// TIA Portal V20 export
// export: Created 2025-12-01T14:56:22.0894666Z, ExportSetting None, DisplayName Totally Integrated Automation Portal, DisplayVersion V20 Update 3, DisplayName TIA Portal Openness, DisplayVersion V20 Update 3, DisplayName TIA Portal Version Control Interface, DisplayVersion V20 Update 3, DisplayName STEP 7 Professional, DisplayVersion V20 Update 3, DisplayName STEP 7 Safety, DisplayVersion V20 Update 2, DisplayName WinCC Basic/Comfort/Advanced, DisplayVersion V20 Update 3, DisplayName WinCC Professional, DisplayVersion V20 Update 3, DisplayName WinCC Unified, DisplayVersion V20 Update 3
TYPE "NDD_Interlock_Horquilla"
   STRUCT
      PosHorq_Bloqueo : Bool;   // La Horquilla esta en Bloqueo para ir a la Posicion IN (Hacia el Elevador)
      MovHorq_Bloqueada : Bool;
      OrdenDeSalida : Bool;   // Orden de la Salida de la Paleta de la Horquilla
      FinOrdenDeSalida : Bool;
      DejarCarga_EntradaHorq : Bool;
      DejadaCarga_EntradaHorq : Bool;   // Aviso de Dejar la Paleta en la Horquilla
      RecogerCarga_SalidaHorq : Bool;   // Aviso de Recoger la Paleta de la Horquilla
      RecogidaCarga_SalidaHorq : Bool;
      AVTF_EntradaHorq : Bool;   // Aviso de Entrada de la Paleta en la Horquilla
      PTF_EntradaHorq : Bool;   // Permiso de Entrada de la Paleta en la Horquilla
      FTF_EntradaHorq : Bool;   // Fin de la Entrada de la Paleta en la Horquilla
      AVTF_SalidaHorq : Bool;   // Aviso de Salida de la Paleta en la Horquilla
      PTF_SalidaHorq : Bool;   // Permiso de Salida de la Paleta en la Hoquilla
      FTF_SalidaHorq : Bool;   // Fin de la Salida de la Paleta en la Hoprquilla
      Libre_16 : Bool;
      DesHabilitarBarrera_Down : Bool;
      ConCarga_Horq : Bool;
      Horq_Out : Bool;
      Horq_In : Bool;
      Horq_SeguridadUp : Bool;
      Horq_SeguridadDown : Bool;
      Libre_25 : Bool;
      Libre_26 : Bool;
      Horq_EnReset : Bool;
      Horq_EnCarga : Bool;
      Horq_EnVacio : Bool;
      Horq_Entrando : Bool;
      Horq_Saliendo : Bool;
      Libre_35 : Bool;
      Libre_36 : Bool;
      Libre_37 : Bool;
   END_STRUCT;
END_TYPE
